FUNCTION_BLOCK ActState (* CAT Function Block Type *)
  (* Standard: 61499-2 *)
  (* Version 0.0, 6/3/2026, Schneider Electric, template *)
  PACKAGE SE.Nereda;
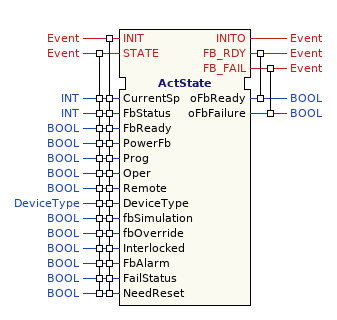
  EVENT_INPUT
    INIT WITH CurrentSp, FbStatus, Prog, Oper, Remote, FbReady, PowerFb, DeviceType, fbSimulation, fbOverride, Interlocked, FbAlarm, FailStatus, NeedReset;
    STATE WITH CurrentSp, FbStatus, FbReady, PowerFb, Prog, Oper, Remote, DeviceType, fbSimulation, fbOverride, Interlocked, FbAlarm, FailStatus, NeedReset;
  END_EVENT
  EVENT_OUTPUT
    INITO;
    FB_RDY WITH oFbReady;
    FB_FAIL WITH oFbFailure;
  END_EVENT
  VAR_INPUT
    CurrentSp : INT;
    FbStatus : INT;
    FbReady : BOOL;
    PowerFb : BOOL;
    Prog : BOOL;
    Oper : BOOL;
    Remote : BOOL;
    DeviceType : DeviceType;
    fbSimulation : BOOL;
    fbOverride : BOOL;
    Interlocked : BOOL;
    FbAlarm : BOOL;
    FailStatus : BOOL;
    NeedReset : BOOL;
  END_VAR
  VAR_OUTPUT
    oFbReady : BOOL;
    oFbFailure : BOOL;
  END_VAR
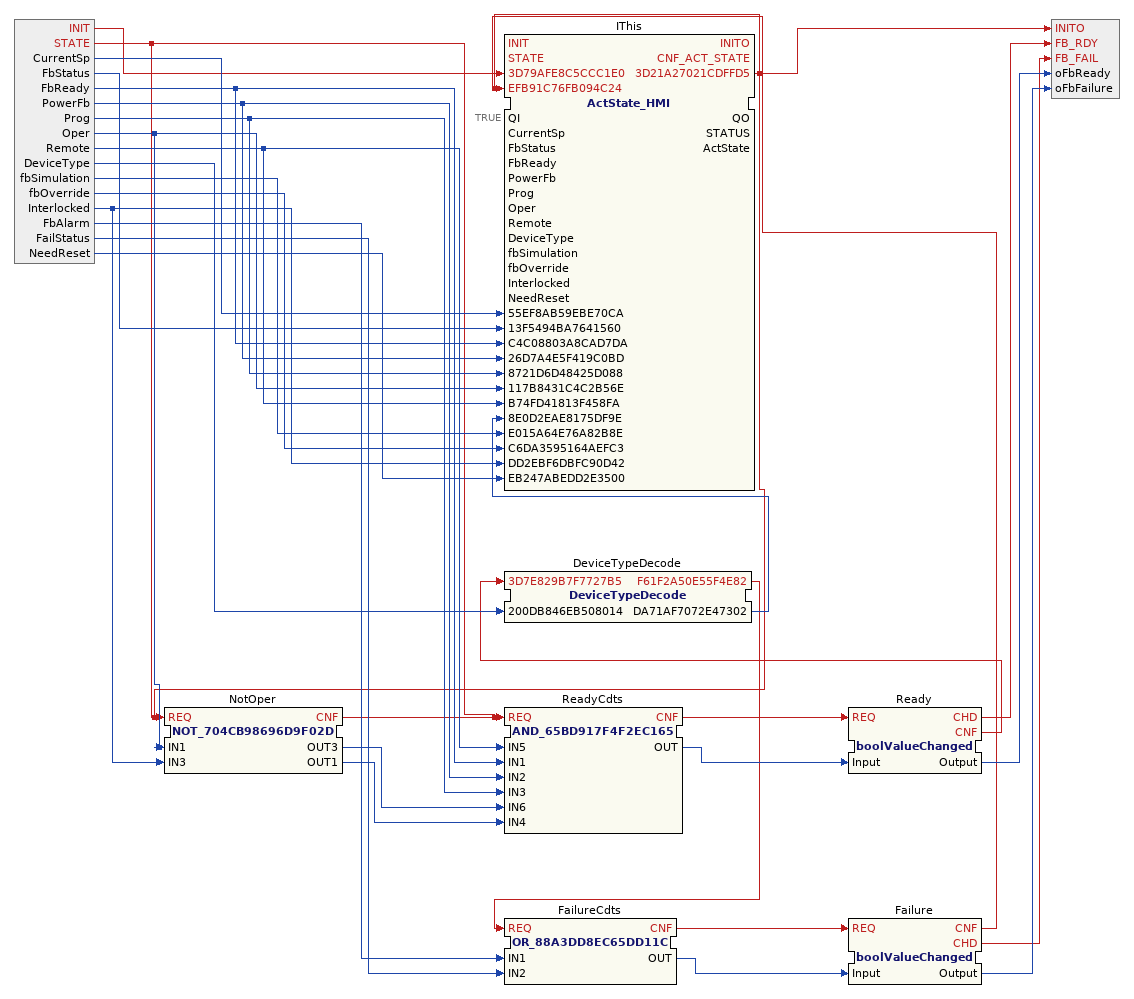
  (* Ready Conditions : Fb Ready = TRUE Fb Power = TRUE Prog = TRUE Oper = FALSE Remote = TRUE Interlock = FALSE *)
  FBS
    IThis : ActState_HMI(QI := TRUE);
    DeviceTypeDecode : DeviceTypeDecode;
    Ready : boolValueChanged;
    ReadyCdts : AND_65BD917F4F2EC165; {SET_ATTRIBUTE(Configuration.GenericFBType.InterfaceParams, Runtime.Standard#CNT:=6;OUT:BOOL)}
    NotOper : NOT_704CB98696D9F02D; {SET_ATTRIBUTE(Configuration.GenericFBType.InterfaceParams, Runtime.Standard#CNT:=3;OUT${CNT$}:BOOL,BOOL,BOOL)}
    FailureCdts : OR_88A3DD8EC65DD11C; {SET_ATTRIBUTE(Configuration.GenericFBType.InterfaceParams, Runtime.Standard#CNT:=2;OUT:BOOL)}
    Failure : boolValueChanged;
  END_FBS
  EVENT_CONNECTIONS
    Ready.CHD TO FB_RDY;
    Ready.CNF TO DeviceTypeDecode.3D7E829B7F7727B5;
    INIT TO IThis.3D79AFE8C5CCC1E0;
    Failure.CNF TO IThis.EFB91C76FB094C24;
    IThis.3D21A27021CDFFD5 TO INITO;
    IThis.3D21A27021CDFFD5 TO IThis.EFB91C76FB094C24;
    STATE TO NotOper.REQ;
    IThis.3D21A27021CDFFD5 TO NotOper.REQ;
    NotOper.CNF TO ReadyCdts.REQ;
    ReadyCdts.CNF TO Ready.REQ;
    Failure.CHD TO FB_FAIL;
    DeviceTypeDecode.F61F2A50E55F4E82 TO FailureCdts.REQ;
    FailureCdts.CNF TO Failure.REQ;
    STATE TO ReadyCdts.REQ;
  END_CONNECTIONS
  DATA_CONNECTIONS
    Ready.Output TO oFbReady;
    DeviceType TO DeviceTypeDecode.200DB846EB508014;
    CurrentSp TO IThis.55EF8AB59EBE70CA;
    FbStatus TO IThis.13F5494BA7641560;
    FbReady TO IThis.C4C08803A8CAD7DA;
    PowerFb TO IThis.26D7A4E5F419C0BD;
    Prog TO IThis.8721D6D48425D088;
    Oper TO IThis.117B8431C4C2B56E;
    Remote TO IThis.B74FD41813F458FA;
    DeviceTypeDecode.DA71AF7072E47302 TO IThis.8E0D2EAE8175DF9E;
    fbSimulation TO IThis.E015A64E76A82B8E;
    fbOverride TO IThis.C6DA3595164AEFC3;
    Interlocked TO IThis.DD2EBF6DBFC90D42;
    Oper TO NotOper.IN1;
    Remote TO ReadyCdts.IN5;
    Interlocked TO NotOper.IN3;
    FbReady TO ReadyCdts.IN1;
    PowerFb TO ReadyCdts.IN2;
    Prog TO ReadyCdts.IN3;
    ReadyCdts.OUT TO Ready.Input;
    NotOper.OUT3 TO ReadyCdts.IN6;
    Failure.Output TO oFbFailure;
    FbAlarm TO FailureCdts.IN1;
    FailStatus TO FailureCdts.IN2;
    FailureCdts.OUT TO Failure.Input;
    NeedReset TO IThis.EB247ABEDD2E3500;
    NotOper.OUT1 TO ReadyCdts.IN4;
  END_CONNECTIONS
END_FUNCTION_BLOCK
